(* Base of Module Sequences. Inheriting FBs must provide the main implementation. *)
FUNCTION_BLOCK ABSTRACT ModuleSequenceBase EXTENDS BehaviorBase
VAR
	m_ptrProcessManager: POINTER TO ProcessManager;
	m_ptrStateTracker: POINTER TO StateTracker;
	m_ptrRaConnector: POINTER TO RaConnector;
END_VAR

METHOD ProvideServices : BOOL
VAR_INPUT
	i_ptrProcessManager: POINTER TO ProcessManager;
	i_ptrStateTracker: POINTER TO StateTracker;
	i_ptrRaConnector: POINTER TO RaConnector;
END_VAR
THIS^.m_ptrProcessManager := i_ptrProcessManager;
THIS^.m_ptrStateTracker := i_ptrStateTracker;
THIS^.m_ptrRaConnector := i_ptrRaConnector;
END_METHOD

METHOD RequestRecovery : BOOL
VAR_INPUT
END_VAR
THIS^.m_ptrRaConnector^.RequestRecovery(THIS^.Postcondition, TO_STRING(m_id));
END_METHOD

END_FUNCTION_BLOCK

(* stored: Version 1.1.0.1, ProductVersion 3.1.4024.12
   POU ModuleSequenceBase: Id {88079229-d709-47ad-8a61-0e1730b237cf}, SpecialFunc None
   Method ProvideServices: Id {7840c96a-62c0-4088-bf67-1e0ef00ed62a}
   Method RequestRecovery: Id {8cc1f64c-bee0-44d7-b390-b6355edc4917} *)
